FUNCTION_BLOCK EL4012
VAR
	_io : EL4xx2_Data;
	{attribute addProperty Name "WcState"}
	_wcState : WcStateBase;
	{attribute addProperty Name "Info data"}
	_infoData : InfoDataAds;
END_VAR

PROPERTY IO : REFERENCE TO EL4xx2_Data
GET
IO REF= _io;
END_GET
END_PROPERTY

PROPERTY WcState : REFERENCE TO WcStateBase
GET
WcState REF= _wcState;
END_GET
END_PROPERTY

END_FUNCTION_BLOCK

(* stored: Version 1.1.0.1, ProductVersion 3.1.4024.9
   POU EL4012: Id {8fe41789-29ec-07a3-21c3-568d316ef8b7}, SpecialFunc None
   Property IO: Id {bec9b823-68b6-085a-3940-bdefd5267082}
   Get Get: Id {fac6456c-504b-05d5-2520-b5e6ed6fea6b}
   Property WcState: Id {bdeee426-7177-0f6a-2700-1b2575bc298f}
   Get Get: Id {0d37bd5e-77da-01e3-3ed6-3fd0f7ec374c} *)
